{attribute 'linkalways'} 
{attribute 'no_explicit_call' := 'This FB is a CLASS and must be accessed using methods or properties'}
{attribute 'enable_dynamic_creation'}
FUNCTION_BLOCK FINAL EQ_DINT EXTENDS Node
VAR
	in1 : _DINT(0);
	in2 : _DINT(0);
	out : _BOOL(FALSE);
END_VAR

METHOD PUBLIC Clone : I_Node
VAR
	pNode : POINTER TO EQ_DINT;
END_VAR
pNode := __NEW(EQ_DINT);
Clone := pNode^;
END_METHOD

METHOD FB_init : BOOL
VAR_INPUT
	bInitRetains : BOOL; // if TRUE, the retain variables are initialized (warm start / cold start)
	bInCopyCode : BOOL;  // if TRUE, the instance afterwards gets moved into the copy code (online change)
END_VAR
AddInput('in1',THIS^.in1);
AddInput('in2',THIS^.in2);
AddOutput('out', THIS^.out);
END_METHOD

METHOD PROTECTED OnExecute
VAR
END_VAR
out.Value := in1.Value = in2.Value;
END_METHOD

END_FUNCTION_BLOCK

(* stored: Version 1.1.0.1, ProductVersion 3.1.4024.15
   POU EQ_DINT: Id {7fa90874-c923-4370-8589-95508582e7df}, SpecialFunc None
   Folder Constructor: Id {1e3ce8f6-fb03-4645-b0ca-75385353738f}
   Method Clone: Id {95062cb7-4cca-498a-b3e4-347bf669909c}
   Method FB_init: Id {c077f883-4901-47cc-a7fa-9180f2a6f98b}
   Method OnExecute: Id {abeda37d-44bd-4474-a478-81a310cd23bc} *)
